{attribute addProperty BoxType "EK1100-0000-0018"}
{attribute addProperty Id "Beckhoff_EL32xxEK1122Beckhoff_EL32xxEK1122_91C4062C162A_0001_EL3201_0000_0016EL3201_FFA6ACB315419.25A_0002_EL3201_0000_0017EL3201_73D65BA516320.375A_0003_EL3201_0000_0018EL3201_73D65BA516320.375A_0004_EL3201_0000_0019EL3201_73D65BA516320.375A_0005_EL3201_0000_0020EL3201_73D65BA516320.375A_0006_EL3201_0000_0021EL3201_73D65BA516320.375A_0007_EL3201_0000_0022EL3201_73D65BA516320.375A_0008_EL3201_0010_0016EL3201_FFA6ACB315419.25A_0009_EL3201_0010_0017EL3201_73D65BA516320.375A_0010_EL3201_0010_0018EL3201_73D65BA516320.375A_0011_EL3201_0010_0019EL3201_73D65BA516320.375A_0012_EL3201_0010_0020EL3201_73D65BA516320.375A_0013_EL3201_0010_0021EL3201_73D65BA516320.375A_0014_EL3201_0010_0022EL3201_73D65BA516320.375A_0015_EL3201_0020_0016EL3201_FFA6ACB315419.25A_0016_EL3201_0020_0017EL3201_73D65BA516320.375A_0017_EL3201_0020_0018EL3201_73D65BA516320.375A_0018_EL3201_0020_0019EL3201_73D65BA516320.375A_0019_EL3201_0020_0020EL3201_73D65BA516320.375A_0020_EL3201_0020_0021EL3201_73D65BA516320.375A_0021_EL3201_0020_0022EL3201_73D65BA516320.375A_0022_EL3202_0000_0016EL3202_DE533F0522628.25A_0023_EL3202_0000_0017EL3202_CEE8F25A24430.5A_0024_EL3202_0000_0018EL3202_CEE8F25A24430.5A_0025_EL3202_0000_0019EL3202_CEE8F25A24430.5A_0026_EL3202_0000_0020EL3202_CEE8F25A24430.5A_0027_EL3202_0000_0021EL3202_CEE8F25A24430.5A_0028_EL3202_0000_0022EL3202_CEE8F25A24430.5A_0029_EL3202_0010_0016EL3202_DE533F0522628.25A_0030_EL3202_0010_0017EL3202_CEE8F25A24430.5A_0031_EL3202_0010_0018EL3202_CEE8F25A24430.5A_0032_EL3202_0010_0019EL3202_CEE8F25A24430.5A_0033_EL3202_0010_0020EL3202_CEE8F25A24430.5A_0034_EL3202_0010_0021EL3202_CEE8F25A24430.5A_0035_EL3202_0010_0022EL3202_CEE8F25A24430.5A_0036_EL3202_0020_0017EL3202_CEE8F25A24430.5A_0037_EL3202_0020_0018EL3202_CEE8F25A24430.5A_0038_EL3202_0020_0019EL3202_CEE8F25A24430.5A_0039_EL3202_0020_0020EL3202_CEE8F25A24430.5A_0040_EL3202_0020_0021EL3202_CEE8F25A24430.5A_0041_EL3202_0020_0022EL3202_CEE8F25A24430.5A_0042_EL3204_0000_0016EL3204_207AEEE037046.25A_0043_EL3204_0000_0017EL3204_C7F08A9440650.75A_0044_EL3204_0000_0018EL3204_C7F08A9440650.75A_0045_EL3204_0000_0019EL3204_C7F08A9440650.75A_0046_EL3204_0000_0020EL3204_C7F08A9440650.75A_0047_EL3204_0000_0021EL3204_C7F08A9440650.75A_0048_EL3204_0162_0016EL3204_4BD7F06321026.25A_0049_EL3204_0162_0017EL3204_4BD7F06321026.25A_0050_EL3204_0162_0018EL3204_4BD7F06321026.25A_0051_EL3204_0162_0019EL3204_4BD7F06321026.25A_0052_EL3204_0200_0016EL3204_712ECA1B21026.25A_0053_EL3204_0200_0017EL3204_712ECA1B21026.25A_0054_EL3204_0200_0018EL3204_712ECA1B21026.25A_0055_EL3208_0000_0017EL3208_F6ED991533842.25A_0056_EL3208_0000_0018EL3208_F6ED991533842.25A_0057_EL3208_0010_0016EL3208_F6ED991533842.25A_0058_EL3214_0000_0016EL3214_712ECA1B21026.25A_0059_EL3214_0000_0017EL3214_712ECA1B21026.25A_0060_EL3214_0090_0016EL3214_712ECA1B21026.25A_0061_EL3218_0000_0016EL3218_F6ED991533842.25A_0062_EL3218_0000_0017EL3218_F6ED991533842.25A_0063_EL3255_0000_0016EL3255_6616AD4624230.25A_0064_EL3255_0000_0017EL3255_11D0319B24230.25A_0065_EL3255_0000_0018EL3255_11D0319B24230.25A_0066_EL3255_0000_0019EL3255_11D0319B24230.25A_0067_EL3255_0000_0020EL3255_6FD6383319424.25A_0068_EL3255_0000_0021EL3255_7B3AD95824230.25A_0069_EL3255_0000_0022EL3255_7B3AD95824230.25A_0070_EL3255_0000_0023EL3255_7B3AD95824230.25"}
{attribute addProperty CRC "1687786308"}
{attribute addProperty SizeInBites "16334"}
{attribute addProperty SizeInBytes "2041.75"}
TYPE Beckhoff_EL32xx_64999344 EXTENDS EK1100_179A0949 :
STRUCT
	{attribute addProperty Name "Beckhoff_EL32xxEK1122"}
	Beckhoff_EL32xxEK1122 : Beckhoff_EL32xxEK1122_91C4062C;
	{attribute addProperty Name "A_0001_EL3201_0000_0016"}
	A_0001_EL3201_0000_0016 : EL3201_FFA6ACB3;
	{attribute addProperty Name "A_0002_EL3201_0000_0017"}
	A_0002_EL3201_0000_0017 : EL3201_73D65BA5;
	{attribute addProperty Name "A_0003_EL3201_0000_0018"}
	A_0003_EL3201_0000_0018 : EL3201_73D65BA5;
	{attribute addProperty Name "A_0004_EL3201_0000_0019"}
	A_0004_EL3201_0000_0019 : EL3201_73D65BA5;
	{attribute addProperty Name "A_0005_EL3201_0000_0020"}
	A_0005_EL3201_0000_0020 : EL3201_73D65BA5;
	{attribute addProperty Name "A_0006_EL3201_0000_0021"}
	A_0006_EL3201_0000_0021 : EL3201_73D65BA5;
	{attribute addProperty Name "A_0007_EL3201_0000_0022"}
	A_0007_EL3201_0000_0022 : EL3201_73D65BA5;
	{attribute addProperty Name "A_0008_EL3201_0010_0016"}
	A_0008_EL3201_0010_0016 : EL3201_FFA6ACB3;
	{attribute addProperty Name "A_0009_EL3201_0010_0017"}
	A_0009_EL3201_0010_0017 : EL3201_73D65BA5;
	{attribute addProperty Name "A_0010_EL3201_0010_0018"}
	A_0010_EL3201_0010_0018 : EL3201_73D65BA5;
	{attribute addProperty Name "A_0011_EL3201_0010_0019"}
	A_0011_EL3201_0010_0019 : EL3201_73D65BA5;
	{attribute addProperty Name "A_0012_EL3201_0010_0020"}
	A_0012_EL3201_0010_0020 : EL3201_73D65BA5;
	{attribute addProperty Name "A_0013_EL3201_0010_0021"}
	A_0013_EL3201_0010_0021 : EL3201_73D65BA5;
	{attribute addProperty Name "A_0014_EL3201_0010_0022"}
	A_0014_EL3201_0010_0022 : EL3201_73D65BA5;
	{attribute addProperty Name "A_0015_EL3201_0020_0016"}
	A_0015_EL3201_0020_0016 : EL3201_FFA6ACB3;
	{attribute addProperty Name "A_0016_EL3201_0020_0017"}
	A_0016_EL3201_0020_0017 : EL3201_73D65BA5;
	{attribute addProperty Name "A_0017_EL3201_0020_0018"}
	A_0017_EL3201_0020_0018 : EL3201_73D65BA5;
	{attribute addProperty Name "A_0018_EL3201_0020_0019"}
	A_0018_EL3201_0020_0019 : EL3201_73D65BA5;
	{attribute addProperty Name "A_0019_EL3201_0020_0020"}
	A_0019_EL3201_0020_0020 : EL3201_73D65BA5;
	{attribute addProperty Name "A_0020_EL3201_0020_0021"}
	A_0020_EL3201_0020_0021 : EL3201_73D65BA5;
	{attribute addProperty Name "A_0021_EL3201_0020_0022"}
	A_0021_EL3201_0020_0022 : EL3201_73D65BA5;
	{attribute addProperty Name "A_0022_EL3202_0000_0016"}
	A_0022_EL3202_0000_0016 : EL3202_DE533F05;
	{attribute addProperty Name "A_0023_EL3202_0000_0017"}
	A_0023_EL3202_0000_0017 : EL3202_CEE8F25A;
	{attribute addProperty Name "A_0024_EL3202_0000_0018"}
	A_0024_EL3202_0000_0018 : EL3202_CEE8F25A;
	{attribute addProperty Name "A_0025_EL3202_0000_0019"}
	A_0025_EL3202_0000_0019 : EL3202_CEE8F25A;
	{attribute addProperty Name "A_0026_EL3202_0000_0020"}
	A_0026_EL3202_0000_0020 : EL3202_CEE8F25A;
	{attribute addProperty Name "A_0027_EL3202_0000_0021"}
	A_0027_EL3202_0000_0021 : EL3202_CEE8F25A;
	{attribute addProperty Name "A_0028_EL3202_0000_0022"}
	A_0028_EL3202_0000_0022 : EL3202_CEE8F25A;
	{attribute addProperty Name "A_0029_EL3202_0010_0016"}
	A_0029_EL3202_0010_0016 : EL3202_DE533F05;
	{attribute addProperty Name "A_0030_EL3202_0010_0017"}
	A_0030_EL3202_0010_0017 : EL3202_CEE8F25A;
	{attribute addProperty Name "A_0031_EL3202_0010_0018"}
	A_0031_EL3202_0010_0018 : EL3202_CEE8F25A;
	{attribute addProperty Name "A_0032_EL3202_0010_0019"}
	A_0032_EL3202_0010_0019 : EL3202_CEE8F25A;
	{attribute addProperty Name "A_0033_EL3202_0010_0020"}
	A_0033_EL3202_0010_0020 : EL3202_CEE8F25A;
	{attribute addProperty Name "A_0034_EL3202_0010_0021"}
	A_0034_EL3202_0010_0021 : EL3202_CEE8F25A;
	{attribute addProperty Name "A_0035_EL3202_0010_0022"}
	A_0035_EL3202_0010_0022 : EL3202_CEE8F25A;
	{attribute addProperty Name "A_0036_EL3202_0020_0017"}
	A_0036_EL3202_0020_0017 : EL3202_CEE8F25A;
	{attribute addProperty Name "A_0037_EL3202_0020_0018"}
	A_0037_EL3202_0020_0018 : EL3202_CEE8F25A;
	{attribute addProperty Name "A_0038_EL3202_0020_0019"}
	A_0038_EL3202_0020_0019 : EL3202_CEE8F25A;
	{attribute addProperty Name "A_0039_EL3202_0020_0020"}
	A_0039_EL3202_0020_0020 : EL3202_CEE8F25A;
	{attribute addProperty Name "A_0040_EL3202_0020_0021"}
	A_0040_EL3202_0020_0021 : EL3202_CEE8F25A;
	{attribute addProperty Name "A_0041_EL3202_0020_0022"}
	A_0041_EL3202_0020_0022 : EL3202_CEE8F25A;
	{attribute addProperty Name "A_0042_EL3204_0000_0016"}
	A_0042_EL3204_0000_0016 : EL3204_207AEEE0;
	{attribute addProperty Name "A_0043_EL3204_0000_0017"}
	A_0043_EL3204_0000_0017 : EL3204_C7F08A94;
	{attribute addProperty Name "A_0044_EL3204_0000_0018"}
	A_0044_EL3204_0000_0018 : EL3204_C7F08A94;
	{attribute addProperty Name "A_0045_EL3204_0000_0019"}
	A_0045_EL3204_0000_0019 : EL3204_C7F08A94;
	{attribute addProperty Name "A_0046_EL3204_0000_0020"}
	A_0046_EL3204_0000_0020 : EL3204_C7F08A94;
	{attribute addProperty Name "A_0047_EL3204_0000_0021"}
	A_0047_EL3204_0000_0021 : EL3204_C7F08A94;
	{attribute addProperty Name "A_0048_EL3204_0162_0016"}
	A_0048_EL3204_0162_0016 : EL3204_4BD7F063;
	{attribute addProperty Name "A_0049_EL3204_0162_0017"}
	A_0049_EL3204_0162_0017 : EL3204_4BD7F063;
	{attribute addProperty Name "A_0050_EL3204_0162_0018"}
	A_0050_EL3204_0162_0018 : EL3204_4BD7F063;
	{attribute addProperty Name "A_0051_EL3204_0162_0019"}
	A_0051_EL3204_0162_0019 : EL3204_4BD7F063;
	{attribute addProperty Name "A_0052_EL3204_0200_0016"}
	A_0052_EL3204_0200_0016 : EL3204_712ECA1B;
	{attribute addProperty Name "A_0053_EL3204_0200_0017"}
	A_0053_EL3204_0200_0017 : EL3204_712ECA1B;
	{attribute addProperty Name "A_0054_EL3204_0200_0018"}
	A_0054_EL3204_0200_0018 : EL3204_712ECA1B;
	{attribute addProperty Name "A_0055_EL3208_0000_0017"}
	A_0055_EL3208_0000_0017 : EL3208_F6ED9915;
	{attribute addProperty Name "A_0056_EL3208_0000_0018"}
	A_0056_EL3208_0000_0018 : EL3208_F6ED9915;
	{attribute addProperty Name "A_0057_EL3208_0010_0016"}
	A_0057_EL3208_0010_0016 : EL3208_F6ED9915;
	{attribute addProperty Name "A_0058_EL3214_0000_0016"}
	A_0058_EL3214_0000_0016 : EL3214_712ECA1B;
	{attribute addProperty Name "A_0059_EL3214_0000_0017"}
	A_0059_EL3214_0000_0017 : EL3214_712ECA1B;
	{attribute addProperty Name "A_0060_EL3214_0090_0016"}
	A_0060_EL3214_0090_0016 : EL3214_712ECA1B;
	{attribute addProperty Name "A_0061_EL3218_0000_0016"}
	A_0061_EL3218_0000_0016 : EL3218_F6ED9915;
	{attribute addProperty Name "A_0062_EL3218_0000_0017"}
	A_0062_EL3218_0000_0017 : EL3218_F6ED9915;
	{attribute addProperty Name "A_0063_EL3255_0000_0016"}
	A_0063_EL3255_0000_0016 : EL3255_6616AD46;
	{attribute addProperty Name "A_0064_EL3255_0000_0017"}
	A_0064_EL3255_0000_0017 : EL3255_11D0319B;
	{attribute addProperty Name "A_0065_EL3255_0000_0018"}
	A_0065_EL3255_0000_0018 : EL3255_11D0319B;
	{attribute addProperty Name "A_0066_EL3255_0000_0019"}
	A_0066_EL3255_0000_0019 : EL3255_11D0319B;
	{attribute addProperty Name "A_0067_EL3255_0000_0020"}
	A_0067_EL3255_0000_0020 : EL3255_6FD63833;
	{attribute addProperty Name "A_0068_EL3255_0000_0021"}
	A_0068_EL3255_0000_0021 : EL3255_7B3AD958;
	{attribute addProperty Name "A_0069_EL3255_0000_0022"}
	A_0069_EL3255_0000_0022 : EL3255_7B3AD958;
	{attribute addProperty Name "A_0070_EL3255_0000_0023"}
	A_0070_EL3255_0000_0023 : EL3255_7B3AD958;
END_STRUCT
END_TYPE

(* stored: Version 1.2.0.0, ProductVersion 3.1.4024.9
   DUT Beckhoff_EL32xx_64999344: Id {cf4f0dc3-0db3-4ae9-bef0-ef732e249a7b} *)
